// TIA Portal V16 export
// export: Created 2021-07-12T14:47:14.6792603Z, ExportSetting WithDefaults, DisplayName Totally Integrated Automation Portal, DisplayVersion V16, DisplayName TIA Portal Version Control Interface, DisplayVersion V16, DisplayName TIA Portal Openness, DisplayVersion V16, DisplayName STEP 7 Professional, DisplayVersion V16, DisplayName STEP 7 Safety, DisplayVersion V16, DisplayName WinCC Professional, DisplayVersion V16
DATA_BLOCK "TestCharacteristics_03"   // DB5003
{ S7_Optimized_Access := 'TRUE' }
FAMILY : SimaHydTO
VERSION : 1.0
// stored: AutoNumber true, DBAccessibleFromOPCUA true, InstanceOfName LSimaHydTO_typeVCharData, InstanceOfType UDT, IsOnlyStoredInLoadMemory false, IsWriteProtectedInAS false
"LSimaHydTO_typeVCharData"
   // VAR
   //    QOutput { S7_SetPoint := 'True'} : Array[0.."LSIMAHYD_VCHAR_POINTS_UPPER_LIMIT"] of Real;
   //    Velocity { S7_SetPoint := 'True'} : Array[0.."LSIMAHYD_VCHAR_POINTS_UPPER_LIMIT"] of Real;
   //    VelocityLimitPositive { S7_SetPoint := 'True'} : Real;
   //    VelocityLimitNegative { S7_SetPoint := 'True'} : Real;
   //    ZeroZonePositive { S7_SetPoint := 'True'} : Real;
   //    ZeroZoneNegative { S7_SetPoint := 'True'} : Real;
   //    MaxIdx { S7_SetPoint := 'True'} : Int;
   //    "Name" { S7_SetPoint := 'True'} : WString[24] := 'TestCharacteristics_03';
   // END_VAR
BEGIN
END_DATA_BLOCK
